{attribute 'GeneratedUsingTerminal: EK1100-0000-0018'}
{attribute addProperty BoxType "EK1100-0000-0018"}
{attribute addProperty Id "Beckhoff_EP5xxxEK1122Beckhoff_EP5xxxEK1122_4DD10B2C313"}
{attribute addProperty CRC "108181556"}
{attribute addProperty Size "313"}
TYPE Beckhoff_EP5xxx_0672B834 EXTENDS EK1100_1FC0878B :
STRUCT
	{attribute addProperty Name "Beckhoff_EP5xxxEK1122"}
	{attribute addProperty PreviousPort "Beckhoff EP5xxx : B"}
	Beckhoff_EP5xxxEK1122 : Beckhoff_EP5xxxEK1122_4DD10B2C;
END_STRUCT
END_TYPE

(* stored: Version 1.2.0.0, ProductVersion 3.1.4024.9
   DUT Beckhoff_EP5xxx_0672B834: Id {17f5df86-d1da-4a3c-8d71-30e888fb426e} *)
